// TIA Portal V21 export
TYPE "Std_stMalfunction"
   STRUCT
      iMalfunctionCode { ExternalVisible := 'False'} : Int;
      iMalfunctionSubCode { ExternalVisible := 'False'} : Int;
      iMalfunctionClassification { ExternalVisible := 'False'} : Int;
      diHours { ExternalVisible := 'False'} : DInt;
      iMinutes { ExternalVisible := 'False'} : Int;
      iSeconds { ExternalVisible := 'False'} : Int;
      iMilliseconds { ExternalVisible := 'False'} : Int;
   END_STRUCT;
END_TYPE
